FUNCTION_BLOCK OverrideV (* Basic Function Block Type *)
  (* Standard: 61499-2 *)
  (* Version 0.0, 6/26/2026, Schneider Electric, Template *)
  PACKAGE SE.Nereda;
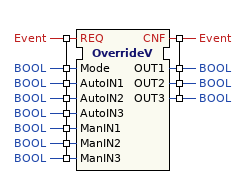
  EVENT_INPUT
    REQ WITH Mode, AutoIN1, AutoIN2, ManIN1, ManIN2, AutoIN3, ManIN3; (* Normal Execution Request *)
  END_EVENT
  EVENT_OUTPUT
    CNF WITH OUT3, OUT1, OUT2; (* Execution Confirmation *)
  END_EVENT
  VAR_INPUT
    Mode : BOOL;
    AutoIN1 : BOOL;
    AutoIN2 : BOOL;
    AutoIN3 : BOOL;
    ManIN1 : BOOL;
    ManIN2 : BOOL;
    ManIN3 : BOOL;
  END_VAR
  VAR_OUTPUT
    OUT1 : BOOL;
    OUT2 : BOOL;
    OUT3 : BOOL;
  END_VAR
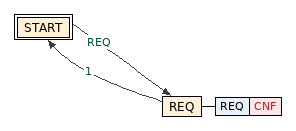
  EC_STATES
    START; (* Initial State *)
    REQ : REQ -> CNF; (* Normal execution *)
  END_STATES
  EC_TRANSITIONS
    START TO REQ := REQ;
    REQ TO START := 1;
  END_TRANSITIONS
  ALGORITHM REQ IN ST: (* Normally executed algorithm *)
;
IF NOT Mode THEN //Auto
	OUT1 := AutoIN1;
	OUT2 := AutoIN2;
	OUT3 := AutoIN3;
ELSIF Mode THEN //Man
	OUT1 := ManIN1;
	OUT2 := ManIN2;
	OUT3 := ManIN3;
END_IF;
  END_ALGORITHM
END_FUNCTION_BLOCK
